/// returns the ADS port number used by the current task
FUNCTION F_GetAdsPort : UINT
VAR
	/// FB to get the index of the current task 
	fbTaskIndex: GETCURTASKINDEX;
END_VAR

fbTaskIndex();
F_GetAdsPort := TwinCAT_SystemInfoVarList._TaskInfo[fbTaskIndex.index].AdsPort;

END_FUNCTION

(* stored: Version 1.1.0.1
   POU F_GetAdsPort: Id {1ec35bb8-a468-4367-a4b9-d8e24742395a}, SpecialFunc None *)
